INTERFACE PUBLIC MotionCommand EXTENDS AsyncCommand

{attribute 'monitoring' := 'call'}
PROPERTY PUBLIC Active : BOOL
GET
END_GET
END_PROPERTY

END_INTERFACE

(* stored: Version 1.1.0.1, ProductVersion 3.1.4026.13
   Itf MotionCommand: Id {8967f49d-aeb8-4635-9a0f-7593c5229e8a}
   Property Active: Id {ec39d927-a338-4482-ac89-2d4222c53c5f}
   Get Get: Id {29c46f42-f1ec-4e59-acd5-5dee44083e27} *)
